// TwinCAT 3 PLC project test01
// ProgramVersion: 3.1.4024.12
// libraries:
//   Tc2_Standard, * (Beckhoff Automation GmbH)
//   Tc2_System, * (Beckhoff Automation GmbH)
//   Tc3_Module, * (Beckhoff Automation GmbH)
// project tree:
//   GVLs/ GVL.TcGVL
//   / PlcTask.TcTTO
//   POUs/ MAIN.TcPOU
// real-time tasks:
//   TASK PlcTask: cycle T#10ms, priority 20, ADS port 350

CONFIGURATION test01
    RESOURCE PLC ON TwinCAT3
        TASK PlcTask(INTERVAL := T#10ms, PRIORITY := 20);
        PROGRAM MAIN WITH PlcTask : MAIN;
    END_RESOURCE
END_CONFIGURATION

// ---- GVLs/GVL.TcGVL
{attribute 'qualified_only'}
VAR_GLOBAL
	DI_00	AT%IX0.0	:BOOL;
	DI_01	AT%IX0.1	:BOOL;
	DI_02	AT%IX0.2	:BOOL;
	DI_03	AT%IX0.3	:BOOL;
	DI_04	AT%IX0.4	:BOOL;
	DI_05	AT%IX0.5	:BOOL;
	DI_06	AT%IX0.6	:BOOL;
	DI_07	AT%IX0.7	:BOOL;
	
	DO_00	AT%QX0.0	:BOOL;
	DO_01	AT%QX0.1	:BOOL;
	DO_02	AT%QX0.2	:BOOL;
	DO_03	AT%QX0.3	:BOOL;
	DO_04	AT%QX0.4	:BOOL;
	DO_05	AT%QX0.5	:BOOL;
	DO_06	AT%QX0.6	:BOOL;
	DO_07	AT%QX0.7	:BOOL;
	
END_VAR

// ---- POUs/MAIN.TcPOU
PROGRAM MAIN
VAR
END_VAR

END_PROGRAM
